FUNCTION_BLOCK FB_Cylinder_NoSensor EXTENDS FB_CylinderBase
VAR_INPUT
END_VAR
VAR_OUTPUT
END_VAR
VAR
END_VAR

METHOD HardwareUpdate : BOOL
VAR_INPUT
END_VAR
fbSimExtend_TON();		//Call timer FB
fbSimRetract_TON();		//Call timer FB

GenerateFeedback(bExtend := bExtendCommand,
				 bRetract := bRetractCommand,
				 bExtended_Generated => bExtendedFeedback,
				 bRetracted_Generated => bRetractedFeedback);
END_METHOD

END_FUNCTION_BLOCK

(* stored: Version 1.1.0.1, ProductVersion 3.1.4024.9
   POU FB_Cylinder_NoSensor: Id {8c5cc0da-3f20-4dda-bfe6-4c6ccc1647cc}, SpecialFunc None
   Folder 01_SUPER_Overrides: Id {a524d52e-6673-48b1-bb0b-410b1f52e431}
   Method HardwareUpdate: Id {e72e7efd-a880-4ee1-acf4-8f52bb9874b2} *)
